PROGRAM Motion
VAR
END_VAR

Motion.StartStop();
Motion.SingleAxis_LD();

METHOD SingleAxis_LD : BOOL
VAR_INPUT
END_VAR
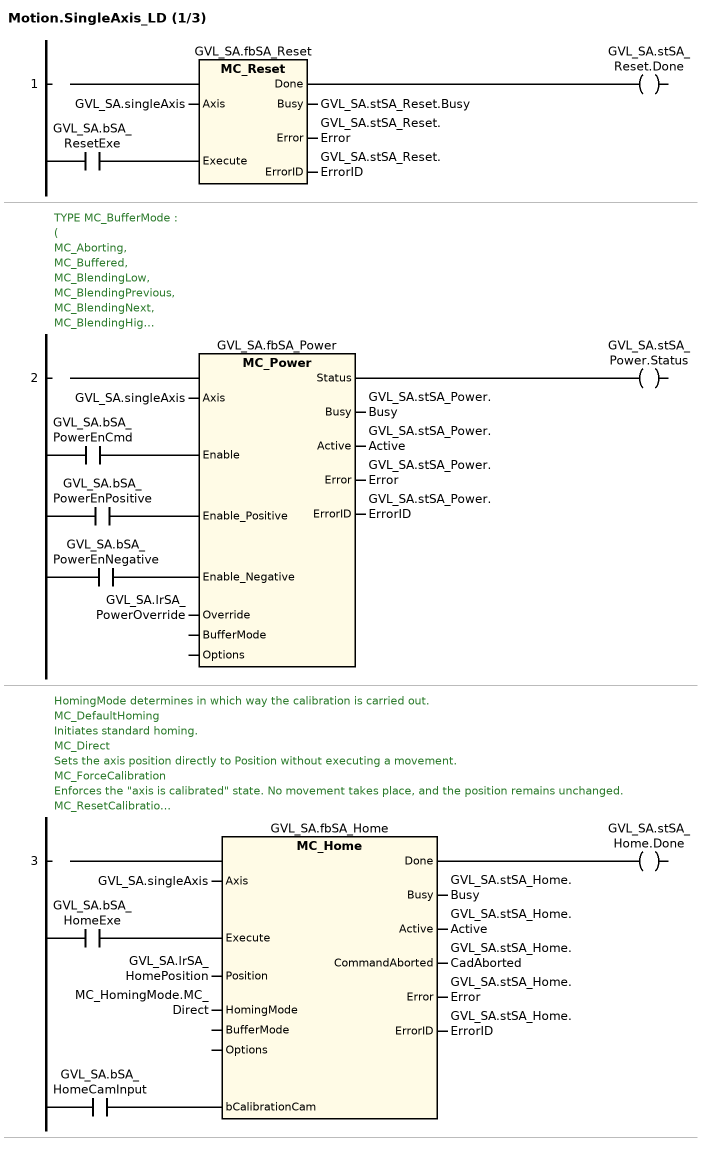
// NETWORK 1
GVL_SA.fbSA_Reset(
    Axis := GVL_SA.singleAxis,
    Execute := GVL_SA.bSA_ResetExe,
    Busy => GVL_SA.stSA_Reset.Busy,
    Error => GVL_SA.stSA_Reset.Error,
    ErrorID => GVL_SA.stSA_Reset.ErrorID); // MC_Reset
GVL_SA.stSA_Reset.Done := GVL_SA.fbSA_Reset.Done;

// NETWORK 2
// TYPE MC_BufferMode :
// (
//     MC_Aborting,
//     MC_Buffered,
//     MC_BlendingLow,
//     MC_BlendingPrevious,
//     MC_BlendingNext,
//     MC_BlendingHigh
// );
// END_TYPE
GVL_SA.fbSA_Power(
    Axis := GVL_SA.singleAxis,
    Enable := GVL_SA.bSA_PowerEnCmd,
    Enable_Positive := GVL_SA.bSA_PowerEnPositive,
    Enable_Negative := GVL_SA.bSA_PowerEnNegative,
    Override := GVL_SA.lrSA_PowerOverride,
    Busy => GVL_SA.stSA_Power.Busy,
    Active => GVL_SA.stSA_Power.Active,
    Error => GVL_SA.stSA_Power.Error,
    ErrorID => GVL_SA.stSA_Power.ErrorID); // MC_Power
GVL_SA.stSA_Power.Status := GVL_SA.fbSA_Power.Status;

// NETWORK 3
// HomingMode determines in which way the calibration is carried out.
//
// MC_DefaultHoming
// Initiates standard homing.
// MC_Direct
// Sets the axis position directly to Position without executing a movement.
// MC_ForceCalibration
// Enforces the "axis is calibrated" state. No movement takes place, and the position remains unchanged.
// MC_ResetCalibration
// Resets the calibration state of the axis. No movement takes place, and the position remains unchanged.
GVL_SA.fbSA_Home(
    Axis := GVL_SA.singleAxis,
    Execute := GVL_SA.bSA_HomeExe,
    Position := GVL_SA.lrSA_HomePosition,
    HomingMode := MC_HomingMode.MC_Direct,
    bCalibrationCam := GVL_SA.bSA_HomeCamInput,
    Busy => GVL_SA.stSA_Home.Busy,
    Active => GVL_SA.stSA_Home.Active,
    CommandAborted => GVL_SA.stSA_Home.CadAborted,
    Error => GVL_SA.stSA_Home.Error,
    ErrorID => GVL_SA.stSA_Home.ErrorID); // MC_Home
GVL_SA.stSA_Home.Done := GVL_SA.fbSA_Home.Done;

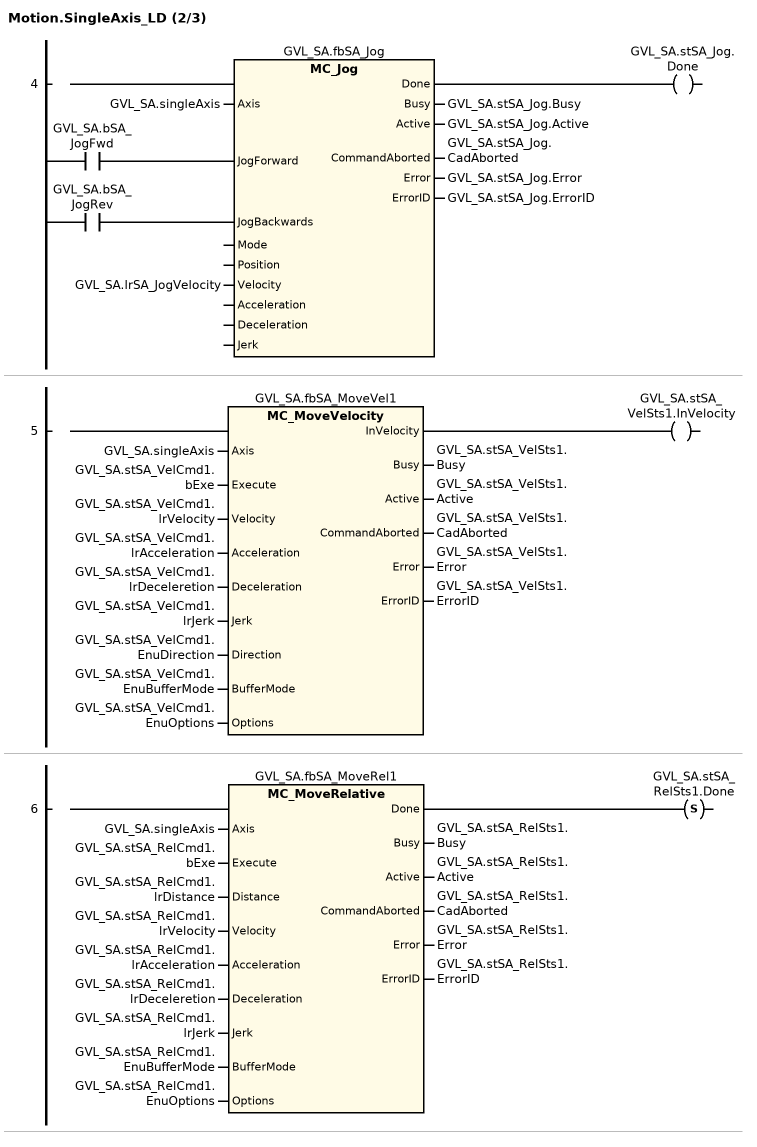
// NETWORK 4
GVL_SA.fbSA_Jog(
    Axis := GVL_SA.singleAxis,
    JogForward := GVL_SA.bSA_JogFwd,
    JogBackwards := GVL_SA.bSA_JogRev,
    Velocity := GVL_SA.lrSA_JogVelocity,
    Busy => GVL_SA.stSA_Jog.Busy,
    Active => GVL_SA.stSA_Jog.Active,
    CommandAborted => GVL_SA.stSA_Jog.CadAborted,
    Error => GVL_SA.stSA_Jog.Error,
    ErrorID => GVL_SA.stSA_Jog.ErrorID); // MC_Jog
GVL_SA.stSA_Jog.Done := GVL_SA.fbSA_Jog.Done;

// NETWORK 5
GVL_SA.fbSA_MoveVel1(
    Axis := GVL_SA.singleAxis,
    Execute := GVL_SA.stSA_VelCmd1.bExe,
    Velocity := GVL_SA.stSA_VelCmd1.lrVelocity,
    Acceleration := GVL_SA.stSA_VelCmd1.lrAcceleration,
    Deceleration := GVL_SA.stSA_VelCmd1.lrDeceleretion,
    Jerk := GVL_SA.stSA_VelCmd1.lrJerk,
    Direction := GVL_SA.stSA_VelCmd1.EnuDirection,
    BufferMode := GVL_SA.stSA_VelCmd1.EnuBufferMode,
    Options := GVL_SA.stSA_VelCmd1.EnuOptions,
    Busy => GVL_SA.stSA_VelSts1.Busy,
    Active => GVL_SA.stSA_VelSts1.Active,
    CommandAborted => GVL_SA.stSA_VelSts1.CadAborted,
    Error => GVL_SA.stSA_VelSts1.Error,
    ErrorID => GVL_SA.stSA_VelSts1.ErrorID); // MC_MoveVelocity
GVL_SA.stSA_VelSts1.InVelocity := GVL_SA.fbSA_MoveVel1.InVelocity;

// NETWORK 6
GVL_SA.fbSA_MoveRel1(
    Axis := GVL_SA.singleAxis,
    Execute := GVL_SA.stSA_RelCmd1.bExe,
    Distance := GVL_SA.stSA_RelCmd1.lrDistance,
    Velocity := GVL_SA.stSA_RelCmd1.lrVelocity,
    Acceleration := GVL_SA.stSA_RelCmd1.lrAcceleration,
    Deceleration := GVL_SA.stSA_RelCmd1.lrDeceleretion,
    Jerk := GVL_SA.stSA_RelCmd1.lrJerk,
    BufferMode := GVL_SA.stSA_RelCmd1.EnuBufferMode,
    Options := GVL_SA.stSA_RelCmd1.EnuOptions,
    Busy => GVL_SA.stSA_RelSts1.Busy,
    Active => GVL_SA.stSA_RelSts1.Active,
    CommandAborted => GVL_SA.stSA_RelSts1.CadAborted,
    Error => GVL_SA.stSA_RelSts1.Error,
    ErrorID => GVL_SA.stSA_RelSts1.ErrorID); // MC_MoveRelative
GVL_SA.stSA_RelSts1.Done S= GVL_SA.fbSA_MoveRel1.Done;

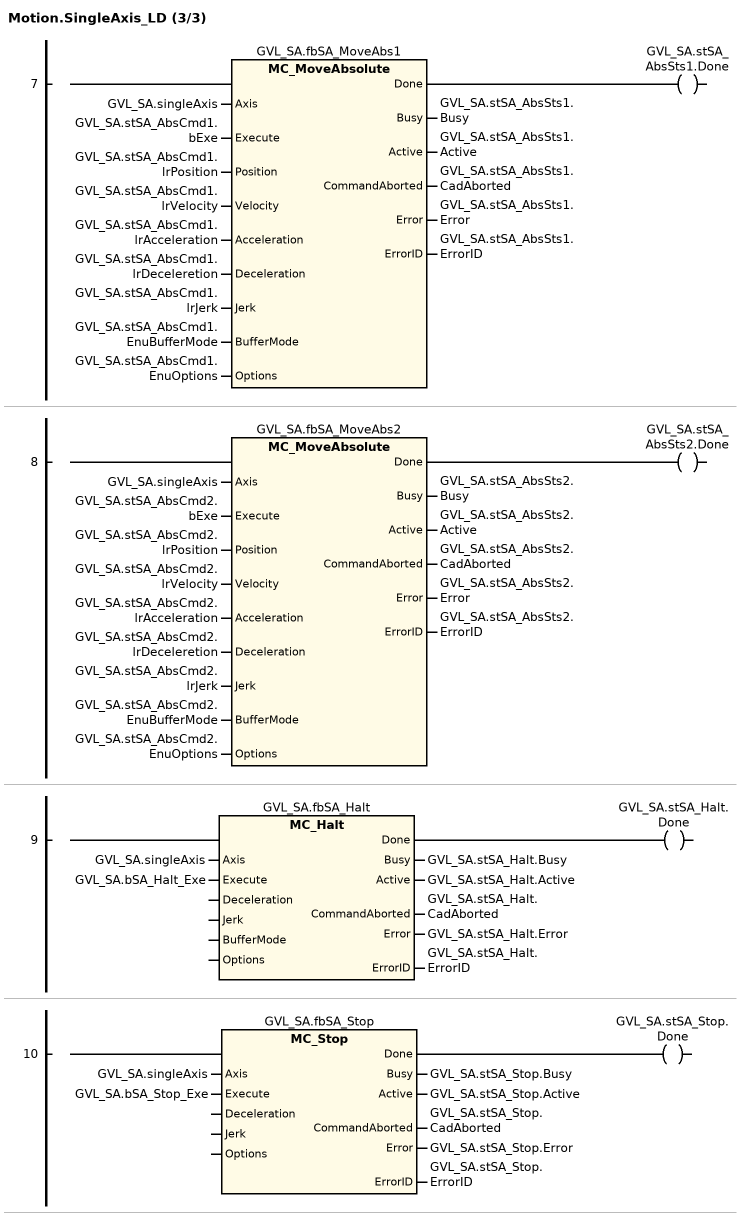
// NETWORK 7
GVL_SA.fbSA_MoveAbs1(
    Axis := GVL_SA.singleAxis,
    Execute := GVL_SA.stSA_AbsCmd1.bExe,
    Position := GVL_SA.stSA_AbsCmd1.lrPosition,
    Velocity := GVL_SA.stSA_AbsCmd1.lrVelocity,
    Acceleration := GVL_SA.stSA_AbsCmd1.lrAcceleration,
    Deceleration := GVL_SA.stSA_AbsCmd1.lrDeceleretion,
    Jerk := GVL_SA.stSA_AbsCmd1.lrJerk,
    BufferMode := GVL_SA.stSA_AbsCmd1.EnuBufferMode,
    Options := GVL_SA.stSA_AbsCmd1.EnuOptions,
    Busy => GVL_SA.stSA_AbsSts1.Busy,
    Active => GVL_SA.stSA_AbsSts1.Active,
    CommandAborted => GVL_SA.stSA_AbsSts1.CadAborted,
    Error => GVL_SA.stSA_AbsSts1.Error,
    ErrorID => GVL_SA.stSA_AbsSts1.ErrorID); // MC_MoveAbsolute
GVL_SA.stSA_AbsSts1.Done := GVL_SA.fbSA_MoveAbs1.Done;

// NETWORK 8
GVL_SA.fbSA_MoveAbs2(
    Axis := GVL_SA.singleAxis,
    Execute := GVL_SA.stSA_AbsCmd2.bExe,
    Position := GVL_SA.stSA_AbsCmd2.lrPosition,
    Velocity := GVL_SA.stSA_AbsCmd2.lrVelocity,
    Acceleration := GVL_SA.stSA_AbsCmd2.lrAcceleration,
    Deceleration := GVL_SA.stSA_AbsCmd2.lrDeceleretion,
    Jerk := GVL_SA.stSA_AbsCmd2.lrJerk,
    BufferMode := GVL_SA.stSA_AbsCmd2.EnuBufferMode,
    Options := GVL_SA.stSA_AbsCmd2.EnuOptions,
    Busy => GVL_SA.stSA_AbsSts2.Busy,
    Active => GVL_SA.stSA_AbsSts2.Active,
    CommandAborted => GVL_SA.stSA_AbsSts2.CadAborted,
    Error => GVL_SA.stSA_AbsSts2.Error,
    ErrorID => GVL_SA.stSA_AbsSts2.ErrorID); // MC_MoveAbsolute
GVL_SA.stSA_AbsSts2.Done := GVL_SA.fbSA_MoveAbs2.Done;

// NETWORK 9
GVL_SA.fbSA_Halt(
    Axis := GVL_SA.singleAxis,
    Execute := GVL_SA.bSA_Halt_Exe,
    Busy => GVL_SA.stSA_Halt.Busy,
    Active => GVL_SA.stSA_Halt.Active,
    CommandAborted => GVL_SA.stSA_Halt.CadAborted,
    Error => GVL_SA.stSA_Halt.Error,
    ErrorID => GVL_SA.stSA_Halt.ErrorID); // MC_Halt
GVL_SA.stSA_Halt.Done := GVL_SA.fbSA_Halt.Done;

// NETWORK 10
GVL_SA.fbSA_Stop(
    Axis := GVL_SA.singleAxis,
    Execute := GVL_SA.bSA_Stop_Exe,
    Busy => GVL_SA.stSA_Stop.Busy,
    Active => GVL_SA.stSA_Stop.Active,
    CommandAborted => GVL_SA.stSA_Stop.CadAborted,
    Error => GVL_SA.stSA_Stop.Error,
    ErrorID => GVL_SA.stSA_Stop.ErrorID); // MC_Stop
GVL_SA.stSA_Stop.Done := GVL_SA.fbSA_Stop.Done;
END_METHOD

METHOD StartStop : BOOL
VAR_INPUT
END_VAR
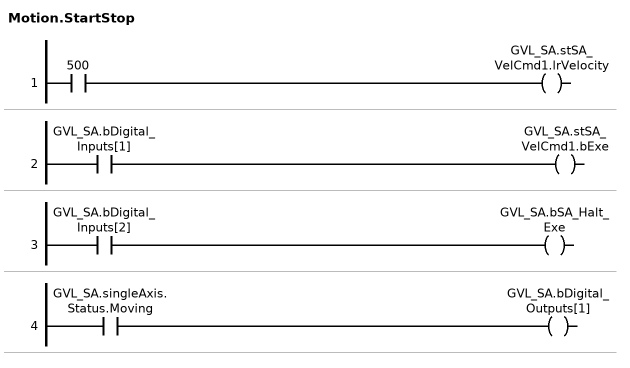
// NETWORK 1
GVL_SA.stSA_VelCmd1.lrVelocity := 500;

// NETWORK 2
GVL_SA.stSA_VelCmd1.bExe := GVL_SA.bDigital_Inputs[1];

// NETWORK 3
GVL_SA.bSA_Halt_Exe := GVL_SA.bDigital_Inputs[2];

// NETWORK 4
GVL_SA.bDigital_Outputs[1] := GVL_SA.singleAxis.Status.Moving;
END_METHOD

END_PROGRAM

(* stored: Version 1.1.0.1, ProductVersion 3.1.4024.12
   POU Motion: Id {9977604b-3578-4d73-9109-4224d81a5e4f}, SpecialFunc None
   Method SingleAxis_LD: Id {0fe1655e-c708-44a8-83ca-6f5316c5a4da}
   Method StartStop: Id {bc71bf8f-a1c5-44f9-b5ff-1454139e1159} *)
